(* PLC project ConveyorLineProject, Schneider Electric EcoStruxure Machine Expert V2.1 *)
(* stored: creationDateTime 2025-09-15T14:30:00, modificationDateTime 2025-09-15T16:45:00 *)

FUNCTION_BLOCK FB_ConveyorControl
  VAR_INPUT
    bStart : BOOL;  (* Start command from HMI *)
    bStop : BOOL;  (* Stop command from HMI *)
    rTargetSpeed : REAL;  (* Target speed in m/min (0..30) *)
    bPhotoEye : BOOL;  (* Product detection photo eye *)
    rMotorCurrent : REAL;  (* Motor current feedback in Amps *)
  END_VAR
  VAR_OUTPUT
    bMotorRun : BOOL;  (* Motor run output to VFD *)
    rSpeedRef : REAL;  (* Speed reference output 0..100% *)
    bJamDetected : BOOL;  (* Jam condition detected *)
    nProductCount : DINT;  (* Products counted since reset *)
    nState : INT;  (* State machine: 0=Idle, 1=Starting, 2=Running, 3=Stopping, 4=Faulted *)
  END_VAR
  VAR
    rCurrentSpeed : REAL;
    rRampRate : REAL := 5.0;
    tJamTimer : TIME;
    tRampTimer : TIME;
    rJamCurrentThreshold : REAL := 15.0;
    bPhotoEyePrev : BOOL;
    aSpeedLog : ARRAY[0..9] OF REAL;  (* Rolling speed log for diagnostics *)
    nLogIndex : INT;
  END_VAR

            (* FB_ConveyorControl - Conveyor belt state machine *)
(* States: 0=Idle, 1=Starting, 2=Running, 3=Stopping, 4=Faulted *)

CASE nState OF
  0: (* Idle *)
    bMotorRun := FALSE;
    rSpeedRef := 0.0;
    IF bStart AND NOT bStop THEN
      nState := 1;
      rCurrentSpeed := 0.0;
    END_IF;

  1: (* Starting - ramp up speed *)
    bMotorRun := TRUE;
    rCurrentSpeed := rCurrentSpeed + rRampRate;
    IF rCurrentSpeed >= rTargetSpeed THEN
      rCurrentSpeed := rTargetSpeed;
      nState := 2;
    END_IF;
    rSpeedRef := (rCurrentSpeed / 30.0) * 100.0;

  2: (* Running *)
    bMotorRun := TRUE;
    rSpeedRef := (rTargetSpeed / 30.0) * 100.0;

    (* Jam detection: motor current exceeds threshold *)
    IF rMotorCurrent > rJamCurrentThreshold THEN
      bJamDetected := TRUE;
      nState := 4;
    END_IF;

    (* Product counting on rising edge of photo eye *)
    IF bPhotoEye AND NOT bPhotoEyePrev THEN
      nProductCount := nProductCount + 1;
    END_IF;
    bPhotoEyePrev := bPhotoEye;

    (* Speed logging for diagnostics *)
    aSpeedLog[nLogIndex] := rCurrentSpeed;
    nLogIndex := (nLogIndex + 1) MOD 10;

    IF bStop THEN
      nState := 3;
    END_IF;

  3: (* Stopping - ramp down *)
    rCurrentSpeed := rCurrentSpeed - rRampRate;
    IF rCurrentSpeed <= 0.0 THEN
      rCurrentSpeed := 0.0;
      bMotorRun := FALSE;
      nState := 0;
    END_IF;
    rSpeedRef := (rCurrentSpeed / 30.0) * 100.0;

  4: (* Faulted *)
    bMotorRun := FALSE;
    rSpeedRef := 0.0;
    (* Require explicit reset via ResetFault action *)
END_CASE;
          
END_FUNCTION_BLOCK

PROGRAM PLC_PRG
  VAR
    fbConveyor1 : FB_ConveyorControl;  (* Infeed conveyor *)
    fbConveyor2 : FB_ConveyorControl;  (* Outfeed conveyor *)
    bSystemReady : BOOL;
    bGlobalEStop : BOOL;
    nTotalProducts : DINT;
    rLineEfficiency : REAL;
    sAlarmText : STRING(120);
    aZoneSpeeds : ARRAY[1..4] OF REAL;
  END_VAR

            (* PLC_PRG - Main cyclic program *)

(* Emergency stop handling *)
IF bGlobalEStop THEN
    fbConveyor1(bStart := FALSE, bStop := TRUE, rTargetSpeed := 0.0,
                bPhotoEye := FALSE, rMotorCurrent := 0.0);
    fbConveyor2(bStart := FALSE, bStop := TRUE, rTargetSpeed := 0.0,
                bPhotoEye := FALSE, rMotorCurrent := 0.0);
    sAlarmText := 'EMERGENCY STOP ACTIVE';
    RETURN;
END_IF;

(* Normal operation: call conveyor function blocks *)
fbConveyor1(rTargetSpeed := aZoneSpeeds[1]);
fbConveyor2(rTargetSpeed := aZoneSpeeds[2]);

(* Aggregate product count *)
nTotalProducts := fbConveyor1.nProductCount + fbConveyor2.nProductCount;

(* System status *)
bSystemReady := NOT bGlobalEStop
                AND NOT fbConveyor1.bJamDetected
                AND NOT fbConveyor2.bJamDetected;

(* Line efficiency calc *)
IF nTotalProducts > 0 THEN
    rLineEfficiency := INT_TO_REAL(nTotalProducts) / 1000.0 * 100.0;
    IF rLineEfficiency > 100.0 THEN
        rLineEfficiency := 100.0;
    END_IF;
END_IF;
          
END_PROGRAM

FUNCTION FC_Hysteresis : BOOL
  VAR_INPUT
    rValue : REAL;  (* Process value to compare *)
    rHighThreshold : REAL;  (* Upper threshold (set point) *)
    rLowThreshold : REAL;  (* Lower threshold (reset point) *)
  END_VAR
  VAR_IN_OUT
    bPreviousState : BOOL;  (* Previous output state (caller must retain) *)
  END_VAR
  VAR
    bResult : BOOL;
  END_VAR

            (* FC_Hysteresis - Hysteresis comparator function *)
(* Once rValue rises above rHighThreshold, output is TRUE.
   Output stays TRUE until rValue falls below rLowThreshold. *)

IF rValue >= rHighThreshold THEN
    bResult := TRUE;
ELSIF rValue <= rLowThreshold THEN
    bResult := FALSE;
ELSE
    bResult := bPreviousState;
END_IF;

bPreviousState := bResult;
FC_Hysteresis := bResult;
          
END_FUNCTION

CONFIGURATION ConveyorLine
  RESOURCE Application ON PLC
    TASK MainTask(INTERVAL := T#10ms, PRIORITY := 1);
    PROGRAM PLC_PRG WITH MainTask : PLC_PRG;
  END_RESOURCE
END_CONFIGURATION
